TYPE ST_Coordinates :
STRUCT
	fX	: LREAL;	// The tag position's x-coordinate in mm.
	fY	: LREAL;	// The tag position's y-coordinate in mm.
	fZ	: LREAL;	// The tag position's z-coordinate in mm.
END_STRUCT
END_TYPE

(* stored: Version 1.1.0.1, ProductVersion 3.1.4024.3
   DUT ST_Coordinates: Id {e6292993-ac8a-4b26-9d0a-074140ebf24c} *)
